// TIA Portal V20 export
TYPE "typeCmInterface"
// stored: Access Published, Namespace Unit1.Em6
   STRUCT
      softcam : "Unit1.Em6.typeCmInterfaceSoftCam";
      brakeTest : "Unit1.Em6.typeCmInterfaceBrakeTest";
   END_STRUCT;
END_TYPE
